// TIA Portal project "Project4" (V18)

(* hardware
DEVICE "S7-1500/ET200MP station_1"  S7-1500 station
   slot 0: "Rail_0"  Rack  6ES7 590-1***0-0AA0
   slot 1: "PLC_1"  CPU 1516F-3 PN/DP  6ES7 516-3FN01-0AB0  V2.9
      slot 3: "CPU display_1"  6ES7591-1BA00-0AA0
      slot 32768: "PROFINET interface_1"  X1
         slot 32769: "Port_1"  X1 P1
         slot 32770: "Port_2"  X1 P2
      slot 33024: "PROFINET interface_2"  X2
         slot 33025: "Port_1"  X2 P1
      slot 33280: "DP interface_1"  X3
      slot 34817: "Virtual CP interface port_1"  Virtual CP interface port  Virtual CP interface port
DEVICE "GSD device_1"  GSD.Device.PN
   slot 0: "Rack"  Rack  V1.0
   slot 0: "UR20-FBC-PN-IRT-V2"  UR20-FBC-PN-IRT-V2 Profinet Device  V01.14.00
      slot 0: "UR20-FBC-PN-IRT-V2 Profinet Device"  UR20-FBC-PN-IRT-V2 Profinet Device
      slot 1: "UR20-FBC-PN-IRT Profinet Device"  UR20-FBC-PN-IRT Profinet Device
         slot 1: "Port 1"  Port 1
         slot 2: "Port 2"  Port 2
   slot 1: "UR20-8DO-P_1"  UR20-8DO-P  1315240000
      slot 0: "UR20-8DO-P"  UR20-8DO-P
   slot 2: "UR20-PF-O-1DI-SIL_1"  UR20-PF-O-1DI-SIL  1335030000
      slot 0: "UR20-PF-O-1DI-SIL"  UR20-PF-O-1DI-SIL
   slot 3: "UR20-16DI-P_1"  UR20-16DI-P  1315200000
      slot 0: "UR20-16DI-P"  UR20-16DI-P
   slot 4: "UR20-4AI-UI-16_1"  UR20-4AI-UI-16  1315620000
      slot 0: "UR20-4AI-UI-16"  UR20-4AI-UI-16
   slot 5: "UR20-4COM-IOL-128BYTE-INOUT_1"  UR20-4COM-IOL-128BYTE-INOUT  1315740000
      slot 0: "UR20-4COM-IOL-128BYTE-INOUT"  UR20-4COM-IOL-128BYTE-INOUT
*)

// ===== PLC "PLC_1"  CPU 1516F-3 PN/DP =====

VAR_GLOBAL   // PLC tag table "Default tag table"
   "UR20_Port0_IN" AT %I16.0 : "DUT_32Bytes";
   "UR20_Port0_OUT" AT %Q16.0 : "DUT_1Bytes";
   "UR20_Port2_OUT" AT %Q17.0 : "DUT_1Bytes";
   "UR20_Port3_OUT" AT %Q18.0 : "DUT_2Bytes";
   "UR20_Port1_IN" AT %I48.0 : "DUT_32Bytes";
   "UR20_Port2_IN" AT %I80.0 : "DUT_32Bytes";
   "UR20_Port3_IN" AT %I112.0 : "DUT_32Bytes";
   "UR20_DIs" AT %I14.0 : "DUT_UR20_DI";
   "UR20_DOs" AT %Q14.0 : "DUT_UR20_DO";
END_VAR

TYPE "DUT_OMRON_E3AS_HL500LMN_IN_Status"
   STRUCT
      ControlOutput1 : Bool;
      ControlOutput2 : Bool;
      InstabilityAlarm : Bool;
      InsufficinetError : Bool;
      Warning : Bool;
      Error : Bool;
   END_STRUCT;
END_TYPE

TYPE "DUT_OMRON_E3AS_HL500LMN_IN"
   STRUCT
      DetectValue : Int;
      LightLevel : Int;
      Status : "DUT_OMRON_E3AS_HL500LMN_IN_Status";
   END_STRUCT;
END_TYPE

TYPE "DUT_NASS_IN"
   STRUCT
      ValveState : Bool;
      ShortCircuit : Bool;
      OpenCircuit : Bool;
      OverHeat : Bool;
      OverCurrent : Bool;
      Counter1OverRun : Bool;
      Counter2OverRun : Bool;
   END_STRUCT;
END_TYPE

TYPE "DUT_NASS_OUT"
   STRUCT
      ON : Bool;
      PWM : Int;
   END_STRUCT;
END_TYPE

TYPE "DUT_OMRON_E2E_X3B4_IL3_2M_IN_Status"
   STRUCT
      Output : Bool;
      Unstable : Bool;
      TooClose : Bool;
      Error : Bool;
   END_STRUCT;
END_TYPE

TYPE "DUT_OMRON_E2E_X3B4_IL3_2M_IN"
   STRUCT
      Montior : Int;
      Status : "DUT_OMRON_E2E_X3B4_IL3_2M_IN_Status";
   END_STRUCT;
END_TYPE

TYPE "DUT_1Bytes"
   STRUCT
      raw : Array[0..0] of Byte;
   END_STRUCT;
END_TYPE

TYPE "DUT_NASS"
   STRUCT
      in : "DUT_NASS_IN";
      out : "DUT_NASS_OUT";
   END_STRUCT;
END_TYPE

TYPE "DUT_2Bytes"
   STRUCT
      raw : Array[0..1] of Byte;
   END_STRUCT;
END_TYPE

TYPE "DUT_4Bytes"
   STRUCT
      raw : Array[0..3] of Byte;
   END_STRUCT;
END_TYPE

TYPE "DUT_32Bytes"
   STRUCT
      raw : Array[0..31] of Byte;
   END_STRUCT;
END_TYPE

TYPE "DUT_UR20_DI"
   STRUCT
      DI1 : Bool;
      DI2 : Bool;
      DI3 : Bool;
      DI4 : Bool;
      CQ1 : Bool;
      CQ2 : Bool;
      CQ3 : Bool;
      CQ4 : Bool;
      ProcessDataInVaildPort1 : Bool;
      ProcessDataInVaildPort2 : Bool;
      ProcessDataInVaildPort3 : Bool;
      ProcessDataInVaildPort4 : Bool;
      ErrorPort1 : Bool;
      ErrorPort2 : Bool;
      ErrorPort3 : Bool;
      ErrorPort4 : Bool;
   END_STRUCT;
END_TYPE

TYPE "DUT_UR20_DO"
   STRUCT
      DO1 : Bool;
      DO2 : Bool;
      DO3 : Bool;
      DO4 : Bool;
      _1 : Bool;
      _2 : Bool;
      _3 : Bool;
      _4 : Bool;
      ProcessDataOutVaildPort1 : Bool;
      ProcessDataOutVaildPort2 : Bool;
      ProcessDataOutVaildPort3 : Bool;
      ProcessDataOutVaildPort4 : Bool;
      _11 : Bool;
      _12 : Bool;
      _13 : Bool;
      _14 : Bool;
   END_STRUCT;
END_TYPE

TYPE "DUT_Murr_59507_OUT"
   STRUCT
      Pin4_X0 : Bool;
      Pin4_X1 : Bool;
      Pin4_X2 : Bool;
      Pin4_X3 : Bool;
      Pin4_X4 : Bool;
      Pin4_X5 : Bool;
      Pin4_X6 : Bool;
      Pin4_X7 : Bool;
   END_STRUCT;
END_TYPE

TYPE "DUT_Murr_59507"
   STRUCT
      in : "DUT_Murr_59507_IN";
      out : "DUT_Murr_59507_OUT";
   END_STRUCT;
END_TYPE

TYPE "DUT_Murr_59507_IN"
   STRUCT
      Pin4_X0 : Bool;
      Pin4_X1 : Bool;
      Pin4_X2 : Bool;
      Pin4_X3 : Bool;
      Pin4_X4 : Bool;
      Pin4_X5 : Bool;
      Pin4_X6 : Bool;
      Pin4_X7 : Bool;
      ErrorPowerSupply : Bool;
      ErrorTemperatureRating : Bool;
      ErrorInputOutput : Bool;
      DIAs : Byte;
      GlobalStatus : Bool;
      DeviceDefine : Byte;
   END_STRUCT;
END_TYPE

DATA_BLOCK "Main_Safety_RTG1_DB"   // DB1, F_DB
{ S7_Optimized_Access := 'TRUE' }
NAME : FUSI
VERSION : 0.1
// stored: InstanceOfName Main_Safety_RTG1
"Main_Safety_RTG1"
BEGIN
END_DATA_BLOCK

DATA_BLOCK "DB_UR20"   // DB2
{ S7_Optimized_Access := 'TRUE' }
VERSION : 0.1
   VAR
      DI : "DUT_UR20_DI";
      "DO" : "DUT_UR20_DO";
      Port0 : "DUT_OMRON_E3AS_HL500LMN_IN";
      Port1 : "DUT_OMRON_E2E_X3B4_IL3_2M_IN";
      Port2 : "DUT_NASS";
      Port3 : "DUT_Murr_59507";
   END_VAR
BEGIN
END_DATA_BLOCK

DATA_BLOCK "FB_UR20_DB"   // DB3
{ S7_Optimized_Access := 'TRUE' }
VERSION : 0.1
// stored: InstanceOfName FB_UR20_IOLINK
"FB_UR20_IOLINK"
BEGIN
END_DATA_BLOCK

DATA_BLOCK "FB_TestFlow_DB"   // DB4
{ S7_Optimized_Access := 'TRUE' }
VERSION : 0.1
// stored: InstanceOfName FB_TestFlow
"FB_TestFlow"
BEGIN
END_DATA_BLOCK

FUNCTION_BLOCK "Main_Safety_RTG1"   // FB1, F_FBD
{ S7_Optimized_Access := 'TRUE' }
BEGIN
END_FUNCTION_BLOCK

FUNCTION_BLOCK "FB_NASS_SmartConnector"   // FB2, LAD
{ S7_Optimized_Access := 'TRUE' }
VERSION : 0.1
   VAR_INPUT
      iEnable : Bool;
   END_VAR
   VAR_IN_OUT
      ioRawIN : Array[*] of Byte;
      ioRawOut : Array[*] of Byte;
      ioData : "DUT_NASS";
   END_VAR
   VAR_TEMP
      _Enable : Bool;
   END_VAR
   VAR_TEMP   // added for the SCL form of the ladder/FBD networks
      _w1 : Bool;
   END_VAR
BEGIN

REGION Network 1
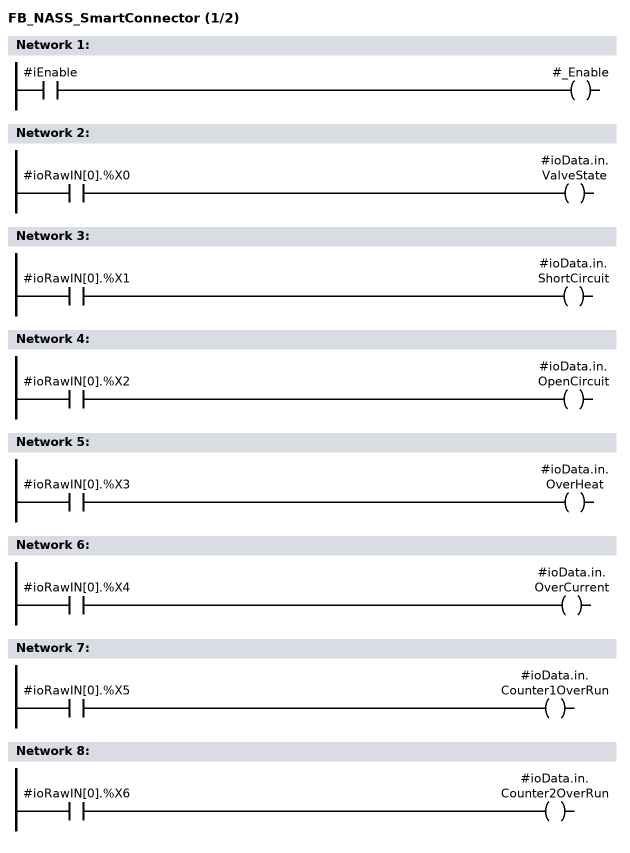
   RUNG wire#powerrail
      Contact( #iEnable )
      Coil( #_Enable )
   END_RUNG
   // the same network as SCL:
   #_Enable := #iEnable;
END_REGION

REGION Network 2
   RUNG wire#powerrail
      Contact( #ioRawIN[0].%X0 )
      Coil( #ioData.in.ValveState )
   END_RUNG
   // the same network as SCL:
   #ioData.in.ValveState := #ioRawIN[0].%X0;
END_REGION

REGION Network 3
   RUNG wire#powerrail
      Contact( #ioRawIN[0].%X1 )
      Coil( #ioData.in.ShortCircuit )
   END_RUNG
   // the same network as SCL:
   #ioData.in.ShortCircuit := #ioRawIN[0].%X1;
END_REGION

REGION Network 4
   RUNG wire#powerrail
      Contact( #ioRawIN[0].%X2 )
      Coil( #ioData.in.OpenCircuit )
   END_RUNG
   // the same network as SCL:
   #ioData.in.OpenCircuit := #ioRawIN[0].%X2;
END_REGION

REGION Network 5
   RUNG wire#powerrail
      Contact( #ioRawIN[0].%X3 )
      Coil( #ioData.in.OverHeat )
   END_RUNG
   // the same network as SCL:
   #ioData.in.OverHeat := #ioRawIN[0].%X3;
END_REGION

REGION Network 6
   RUNG wire#powerrail
      Contact( #ioRawIN[0].%X4 )
      Coil( #ioData.in.OverCurrent )
   END_RUNG
   // the same network as SCL:
   #ioData.in.OverCurrent := #ioRawIN[0].%X4;
END_REGION

REGION Network 7
   RUNG wire#powerrail
      Contact( #ioRawIN[0].%X5 )
      Coil( #ioData.in.Counter1OverRun )
   END_RUNG
   // the same network as SCL:
   #ioData.in.Counter1OverRun := #ioRawIN[0].%X5;
END_REGION

REGION Network 8
   RUNG wire#powerrail
      Contact( #ioRawIN[0].%X6 )
      Coil( #ioData.in.Counter2OverRun )
   END_RUNG
   // the same network as SCL:
   #ioData.in.Counter2OverRun := #ioRawIN[0].%X6;
END_REGION

REGION Network 9
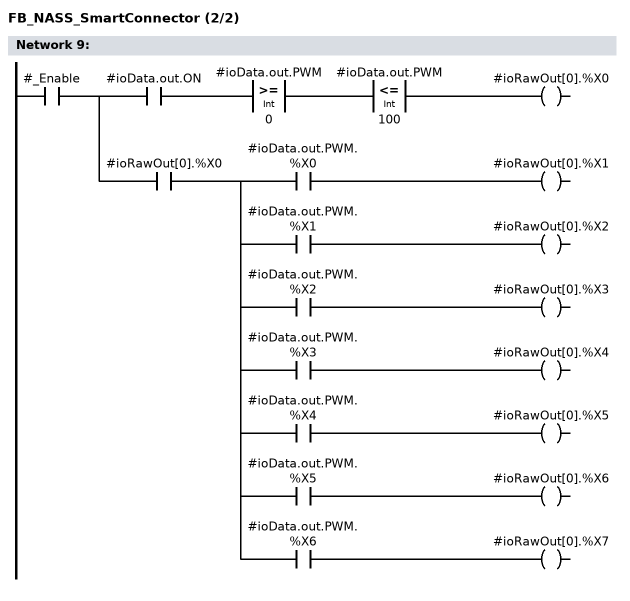
   RUNG wire#powerrail
      Contact( #_Enable )
      wire#w1
      Contact( #ioData.out.ON )
      { S7_Templates := "SrcType := Int" } GE_Contact(in1 := #ioData.out.PWM, in2 := 0)
      { S7_Templates := "SrcType := Int" } LE_Contact(in1 := #ioData.out.PWM, in2 := 100)
      Coil( #ioRawOut[0].%X0 )
   END_RUNG
   RUNG wire#w1
      Contact( #ioRawOut[0].%X0 )
      wire#w2
      Contact( #ioData.out.PWM.%X0 )
      Coil( #ioRawOut[0].%X1 )
   END_RUNG
   RUNG wire#w2
      Contact( #ioData.out.PWM.%X1 )
      Coil( #ioRawOut[0].%X2 )
   END_RUNG
   RUNG wire#w2
      Contact( #ioData.out.PWM.%X2 )
      Coil( #ioRawOut[0].%X3 )
   END_RUNG
   RUNG wire#w2
      Contact( #ioData.out.PWM.%X3 )
      Coil( #ioRawOut[0].%X4 )
   END_RUNG
   RUNG wire#w2
      Contact( #ioData.out.PWM.%X4 )
      Coil( #ioRawOut[0].%X5 )
   END_RUNG
   RUNG wire#w2
      Contact( #ioData.out.PWM.%X5 )
      Coil( #ioRawOut[0].%X6 )
   END_RUNG
   RUNG wire#w2
      Contact( #ioData.out.PWM.%X6 )
      Coil( #ioRawOut[0].%X7 )
   END_RUNG
   // the same network as SCL:
   #ioRawOut[0].%X0 := #_Enable AND #ioData.out.ON AND (#ioData.out.PWM >= 0) AND (#ioData.out.PWM <= 100);
   #_w1 := #_Enable AND #ioRawOut[0].%X0;
   #ioRawOut[0].%X1 := #_w1 AND #ioData.out.PWM.%X0;
   #ioRawOut[0].%X2 := #_w1 AND #ioData.out.PWM.%X1;
   #ioRawOut[0].%X3 := #_w1 AND #ioData.out.PWM.%X2;
   #ioRawOut[0].%X4 := #_w1 AND #ioData.out.PWM.%X3;
   #ioRawOut[0].%X5 := #_w1 AND #ioData.out.PWM.%X4;
   #ioRawOut[0].%X6 := #_w1 AND #ioData.out.PWM.%X5;
   #ioRawOut[0].%X7 := #_w1 AND #ioData.out.PWM.%X6;
END_REGION
END_FUNCTION_BLOCK

FUNCTION_BLOCK "FB_UR20_IOLINK"   // FB3, LAD
{ S7_Optimized_Access := 'TRUE' }
VERSION : 0.1
   VAR
      NassConnector : "FB_NASS_SmartConnector";
      Murr59507 : "FB_Murr_59507";
      OMRONE3ASHL500LMN : "FB_OMRON_E3AS_HL500LMN";
      OMRONE2EX3B4IL32M : "FB_OMRON_E2E_X3B4_IL3_2M";
   END_VAR
   VAR_TEMP
      _temp : Array[0..1] of Byte;
   END_VAR
BEGIN

REGION Network 1
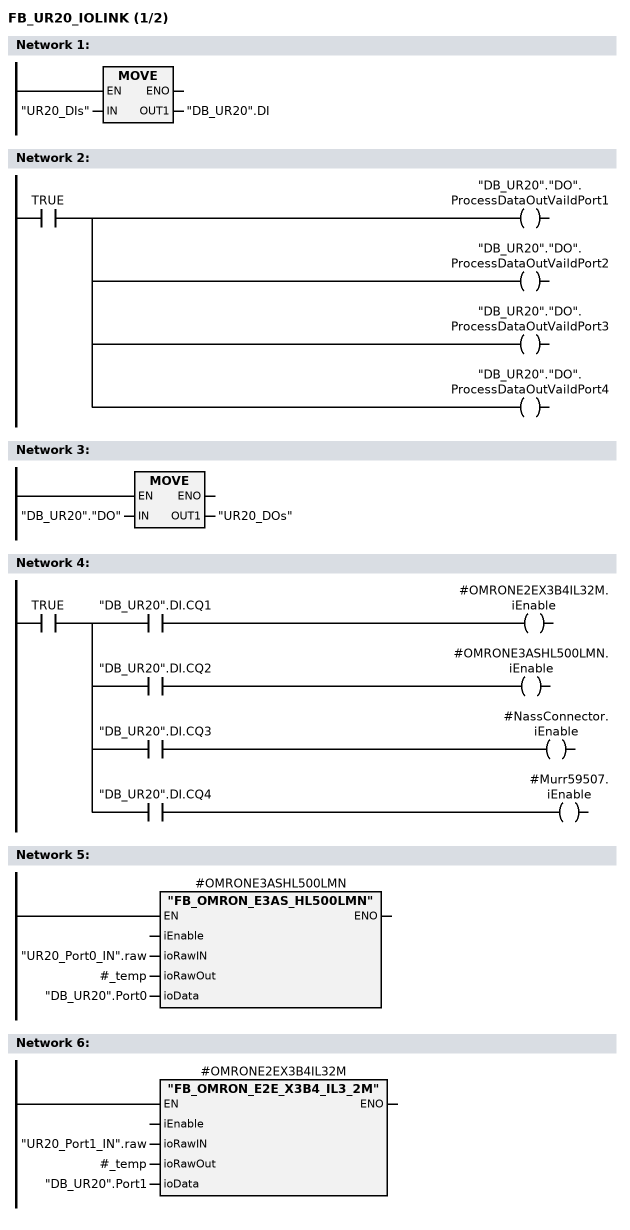
   RUNG wire#powerrail
      Move(in := "UR20_DIs", out1 => "DB_UR20".DI)
   END_RUNG
   // the same network as SCL:
   "DB_UR20".DI := "UR20_DIs";
END_REGION

REGION Network 2
   RUNG wire#powerrail
      Contact( TRUE )
      wire#w1
      Coil( "DB_UR20"."DO".ProcessDataOutVaildPort1 )
   END_RUNG
   RUNG wire#w1
      Coil( "DB_UR20"."DO".ProcessDataOutVaildPort2 )
   END_RUNG
   RUNG wire#w1
      Coil( "DB_UR20"."DO".ProcessDataOutVaildPort3 )
   END_RUNG
   RUNG wire#w1
      Coil( "DB_UR20"."DO".ProcessDataOutVaildPort4 )
   END_RUNG
   // the same network as SCL:
   "DB_UR20"."DO".ProcessDataOutVaildPort1 := TRUE;
   "DB_UR20"."DO".ProcessDataOutVaildPort2 := TRUE;
   "DB_UR20"."DO".ProcessDataOutVaildPort3 := TRUE;
   "DB_UR20"."DO".ProcessDataOutVaildPort4 := TRUE;
END_REGION

REGION Network 3
   RUNG wire#powerrail
      Move(in := "DB_UR20"."DO", out1 => "UR20_DOs")
   END_RUNG
   // the same network as SCL:
   "UR20_DOs" := "DB_UR20"."DO";
END_REGION

REGION Network 4
   RUNG wire#powerrail
      Contact( TRUE )
      wire#w1
      Contact( "DB_UR20".DI.CQ1 )
      Coil( #OMRONE2EX3B4IL32M.iEnable )
   END_RUNG
   RUNG wire#w1
      Contact( "DB_UR20".DI.CQ2 )
      Coil( #OMRONE3ASHL500LMN.iEnable )
   END_RUNG
   RUNG wire#w1
      Contact( "DB_UR20".DI.CQ3 )
      Coil( #NassConnector.iEnable )
   END_RUNG
   RUNG wire#w1
      Contact( "DB_UR20".DI.CQ4 )
      Coil( #Murr59507.iEnable )
   END_RUNG
   // the same network as SCL:
   #OMRONE2EX3B4IL32M.iEnable := TRUE AND "DB_UR20".DI.CQ1;
   #OMRONE3ASHL500LMN.iEnable := TRUE AND "DB_UR20".DI.CQ2;
   #NassConnector.iEnable := TRUE AND "DB_UR20".DI.CQ3;
   #Murr59507.iEnable := TRUE AND "DB_UR20".DI.CQ4;
END_REGION

REGION Network 5
   RUNG wire#powerrail
      #OMRONE3ASHL500LMN(iEnable :=, ioRawIN := "UR20_Port0_IN".raw, ioRawOut := #_temp, ioData := "DB_UR20".Port0)
   END_RUNG
   // the same network as SCL:
   #OMRONE3ASHL500LMN(ioRawIN := "UR20_Port0_IN".raw, ioRawOut := #_temp, ioData := "DB_UR20".Port0);   // "FB_OMRON_E3AS_HL500LMN"
END_REGION

REGION Network 6
   RUNG wire#powerrail
      #OMRONE2EX3B4IL32M(iEnable :=, ioRawIN := "UR20_Port1_IN".raw, ioRawOut := #_temp, ioData := "DB_UR20".Port1)
   END_RUNG
   // the same network as SCL:
   #OMRONE2EX3B4IL32M(ioRawIN := "UR20_Port1_IN".raw, ioRawOut := #_temp, ioData := "DB_UR20".Port1);   // "FB_OMRON_E2E_X3B4_IL3_2M"
END_REGION

REGION Network 7
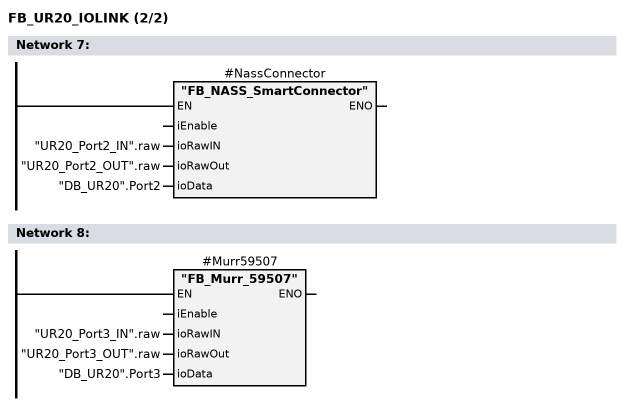
   RUNG wire#powerrail
      #NassConnector(iEnable :=, ioRawIN := "UR20_Port2_IN".raw, ioRawOut := "UR20_Port2_OUT".raw, ioData := "DB_UR20".Port2)
   END_RUNG
   // the same network as SCL:
   #NassConnector(ioRawIN := "UR20_Port2_IN".raw, ioRawOut := "UR20_Port2_OUT".raw, ioData := "DB_UR20".Port2);   // "FB_NASS_SmartConnector"
END_REGION

REGION Network 8
   RUNG wire#powerrail
      #Murr59507(iEnable :=, ioRawIN := "UR20_Port3_IN".raw, ioRawOut := "UR20_Port3_OUT".raw, ioData := "DB_UR20".Port3)
   END_RUNG
   // the same network as SCL:
   #Murr59507(ioRawIN := "UR20_Port3_IN".raw, ioRawOut := "UR20_Port3_OUT".raw, ioData := "DB_UR20".Port3);   // "FB_Murr_59507"
END_REGION
END_FUNCTION_BLOCK

FUNCTION_BLOCK "FB_Murr_59507"   // FB4, LAD
{ S7_Optimized_Access := 'TRUE' }
VERSION : 0.1
   VAR_INPUT
      iEnable : Bool := false;
   END_VAR
   VAR_IN_OUT
      ioRawIN : Array[*] of Byte;
      ioRawOut : Array[*] of Byte;
      ioData : "DUT_Murr_59507";
   END_VAR
   VAR_TEMP
      _Enable : Bool;
   END_VAR
   VAR CONSTANT
      AlwaysON : Bool := 1;
   END_VAR
BEGIN

REGION Network 1
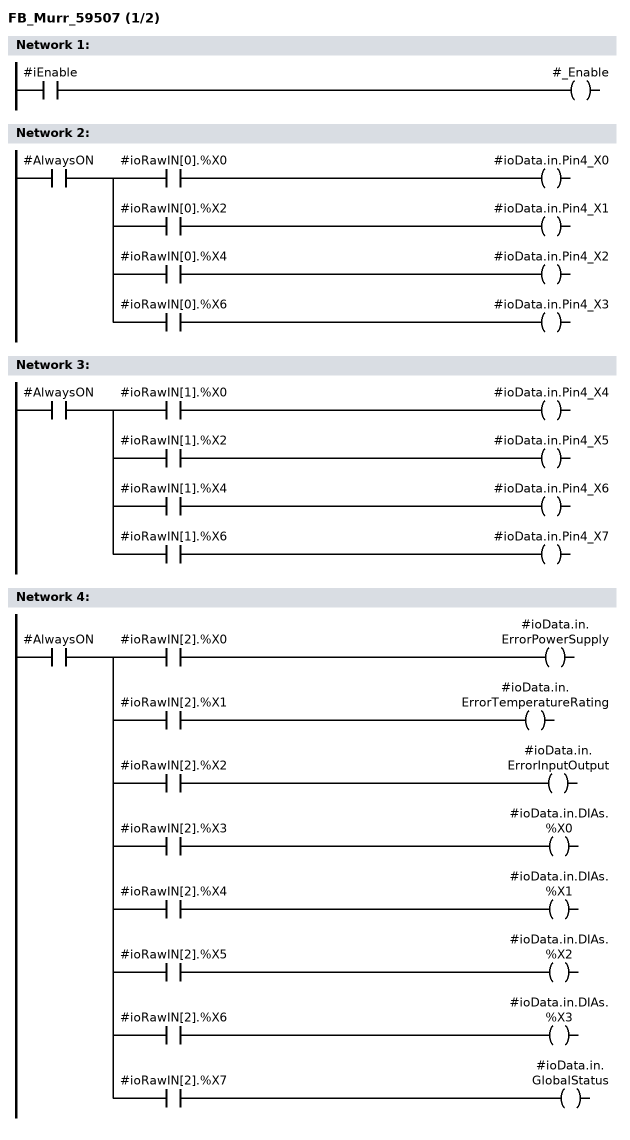
   RUNG wire#powerrail
      Contact( #iEnable )
      Coil( #_Enable )
   END_RUNG
   // the same network as SCL:
   #_Enable := #iEnable;
END_REGION

REGION Network 2
   RUNG wire#powerrail
      Contact( #AlwaysON )
      wire#w1
      Contact( #ioRawIN[0].%X0 )
      Coil( #ioData.in.Pin4_X0 )
   END_RUNG
   RUNG wire#w1
      Contact( #ioRawIN[0].%X2 )
      Coil( #ioData.in.Pin4_X1 )
   END_RUNG
   RUNG wire#w1
      Contact( #ioRawIN[0].%X4 )
      Coil( #ioData.in.Pin4_X2 )
   END_RUNG
   RUNG wire#w1
      Contact( #ioRawIN[0].%X6 )
      Coil( #ioData.in.Pin4_X3 )
   END_RUNG
   // the same network as SCL:
   #ioData.in.Pin4_X0 := #AlwaysON AND #ioRawIN[0].%X0;
   #ioData.in.Pin4_X1 := #AlwaysON AND #ioRawIN[0].%X2;
   #ioData.in.Pin4_X2 := #AlwaysON AND #ioRawIN[0].%X4;
   #ioData.in.Pin4_X3 := #AlwaysON AND #ioRawIN[0].%X6;
END_REGION

REGION Network 3
   RUNG wire#powerrail
      Contact( #AlwaysON )
      wire#w1
      Contact( #ioRawIN[1].%X0 )
      Coil( #ioData.in.Pin4_X4 )
   END_RUNG
   RUNG wire#w1
      Contact( #ioRawIN[1].%X2 )
      Coil( #ioData.in.Pin4_X5 )
   END_RUNG
   RUNG wire#w1
      Contact( #ioRawIN[1].%X4 )
      Coil( #ioData.in.Pin4_X6 )
   END_RUNG
   RUNG wire#w1
      Contact( #ioRawIN[1].%X6 )
      Coil( #ioData.in.Pin4_X7 )
   END_RUNG
   // the same network as SCL:
   #ioData.in.Pin4_X4 := #AlwaysON AND #ioRawIN[1].%X0;
   #ioData.in.Pin4_X5 := #AlwaysON AND #ioRawIN[1].%X2;
   #ioData.in.Pin4_X6 := #AlwaysON AND #ioRawIN[1].%X4;
   #ioData.in.Pin4_X7 := #AlwaysON AND #ioRawIN[1].%X6;
END_REGION

REGION Network 4
   RUNG wire#powerrail
      Contact( #AlwaysON )
      wire#w1
      Contact( #ioRawIN[2].%X0 )
      Coil( #ioData.in.ErrorPowerSupply )
   END_RUNG
   RUNG wire#w1
      Contact( #ioRawIN[2].%X1 )
      Coil( #ioData.in.ErrorTemperatureRating )
   END_RUNG
   RUNG wire#w1
      Contact( #ioRawIN[2].%X2 )
      Coil( #ioData.in.ErrorInputOutput )
   END_RUNG
   RUNG wire#w1
      Contact( #ioRawIN[2].%X3 )
      Coil( #ioData.in.DIAs.%X0 )
   END_RUNG
   RUNG wire#w1
      Contact( #ioRawIN[2].%X4 )
      Coil( #ioData.in.DIAs.%X1 )
   END_RUNG
   RUNG wire#w1
      Contact( #ioRawIN[2].%X5 )
      Coil( #ioData.in.DIAs.%X2 )
   END_RUNG
   RUNG wire#w1
      Contact( #ioRawIN[2].%X6 )
      Coil( #ioData.in.DIAs.%X3 )
   END_RUNG
   RUNG wire#w1
      Contact( #ioRawIN[2].%X7 )
      Coil( #ioData.in.GlobalStatus )
   END_RUNG
   // the same network as SCL:
   #ioData.in.ErrorPowerSupply := #AlwaysON AND #ioRawIN[2].%X0;
   #ioData.in.ErrorTemperatureRating := #AlwaysON AND #ioRawIN[2].%X1;
   #ioData.in.ErrorInputOutput := #AlwaysON AND #ioRawIN[2].%X2;
   #ioData.in.DIAs.%X0 := #AlwaysON AND #ioRawIN[2].%X3;
   #ioData.in.DIAs.%X1 := #AlwaysON AND #ioRawIN[2].%X4;
   #ioData.in.DIAs.%X2 := #AlwaysON AND #ioRawIN[2].%X5;
   #ioData.in.DIAs.%X3 := #AlwaysON AND #ioRawIN[2].%X6;
   #ioData.in.GlobalStatus := #AlwaysON AND #ioRawIN[2].%X7;
END_REGION

REGION Network 5
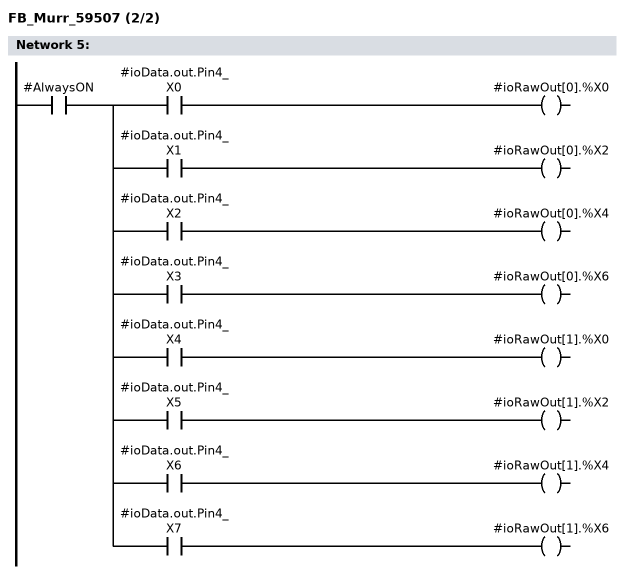
   RUNG wire#powerrail
      Contact( #AlwaysON )
      wire#w1
      Contact( #ioData.out.Pin4_X0 )
      Coil( #ioRawOut[0].%X0 )
   END_RUNG
   RUNG wire#w1
      Contact( #ioData.out.Pin4_X1 )
      Coil( #ioRawOut[0].%X2 )
   END_RUNG
   RUNG wire#w1
      Contact( #ioData.out.Pin4_X2 )
      Coil( #ioRawOut[0].%X4 )
   END_RUNG
   RUNG wire#w1
      Contact( #ioData.out.Pin4_X3 )
      Coil( #ioRawOut[0].%X6 )
   END_RUNG
   RUNG wire#w1
      Contact( #ioData.out.Pin4_X4 )
      Coil( #ioRawOut[1].%X0 )
   END_RUNG
   RUNG wire#w1
      Contact( #ioData.out.Pin4_X5 )
      Coil( #ioRawOut[1].%X2 )
   END_RUNG
   RUNG wire#w1
      Contact( #ioData.out.Pin4_X6 )
      Coil( #ioRawOut[1].%X4 )
   END_RUNG
   RUNG wire#w1
      Contact( #ioData.out.Pin4_X7 )
      Coil( #ioRawOut[1].%X6 )
   END_RUNG
   // the same network as SCL:
   #ioRawOut[0].%X0 := #AlwaysON AND #ioData.out.Pin4_X0;
   #ioRawOut[0].%X2 := #AlwaysON AND #ioData.out.Pin4_X1;
   #ioRawOut[0].%X4 := #AlwaysON AND #ioData.out.Pin4_X2;
   #ioRawOut[0].%X6 := #AlwaysON AND #ioData.out.Pin4_X3;
   #ioRawOut[1].%X0 := #AlwaysON AND #ioData.out.Pin4_X4;
   #ioRawOut[1].%X2 := #AlwaysON AND #ioData.out.Pin4_X5;
   #ioRawOut[1].%X4 := #AlwaysON AND #ioData.out.Pin4_X6;
   #ioRawOut[1].%X6 := #AlwaysON AND #ioData.out.Pin4_X7;
END_REGION
END_FUNCTION_BLOCK

FUNCTION_BLOCK "FB_OMRON_E3AS_HL500LMN"   // FB5, LAD
{ S7_Optimized_Access := 'TRUE' }
VERSION : 0.1
   VAR_INPUT
      iEnable : Bool;
   END_VAR
   VAR_IN_OUT
      ioRawIN : Array[*] of Byte;
      ioRawOut : Array[*] of Byte;
      ioData : "DUT_OMRON_E3AS_HL500LMN_IN";
   END_VAR
   VAR_TEMP
      _Enable : Bool;
   END_VAR
   VAR CONSTANT
      AlwaysON : Bool := 1;
   END_VAR
BEGIN

REGION Network 1
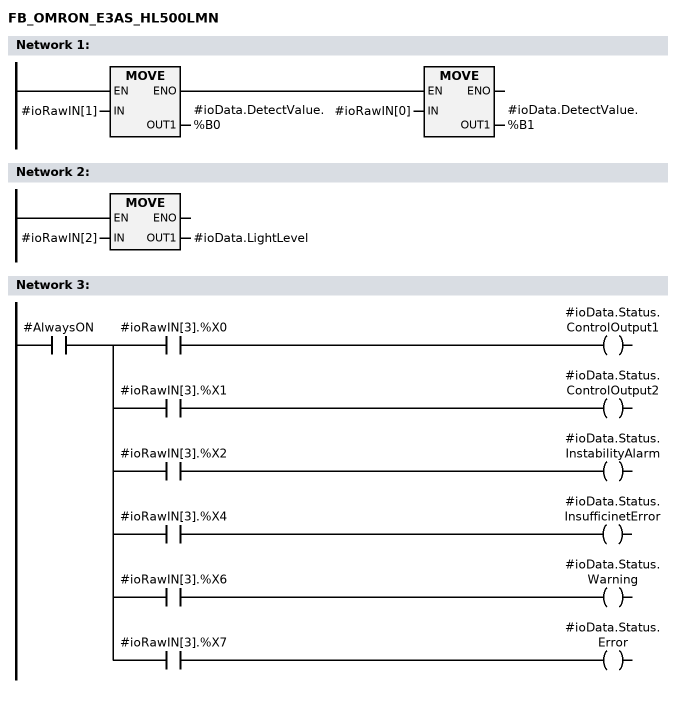
   RUNG wire#powerrail
      Move(in := #ioRawIN[1], out1 => #ioData.DetectValue.%B0)
      Move(in := #ioRawIN[0], out1 => #ioData.DetectValue.%B1)
   END_RUNG
   // the same network as SCL:
   #ioData.DetectValue.%B0 := #ioRawIN[1];
   #ioData.DetectValue.%B1 := #ioRawIN[0];
END_REGION

REGION Network 2
   RUNG wire#powerrail
      Move(in := #ioRawIN[2], out1 => #ioData.LightLevel)
   END_RUNG
   // the same network as SCL:
   #ioData.LightLevel := #ioRawIN[2];
END_REGION

REGION Network 3
   RUNG wire#powerrail
      Contact( #AlwaysON )
      wire#w1
      Contact( #ioRawIN[3].%X0 )
      Coil( #ioData.Status.ControlOutput1 )
   END_RUNG
   RUNG wire#w1
      Contact( #ioRawIN[3].%X1 )
      Coil( #ioData.Status.ControlOutput2 )
   END_RUNG
   RUNG wire#w1
      Contact( #ioRawIN[3].%X2 )
      Coil( #ioData.Status.InstabilityAlarm )
   END_RUNG
   RUNG wire#w1
      Contact( #ioRawIN[3].%X4 )
      Coil( #ioData.Status.InsufficinetError )
   END_RUNG
   RUNG wire#w1
      Contact( #ioRawIN[3].%X6 )
      Coil( #ioData.Status.Warning )
   END_RUNG
   RUNG wire#w1
      Contact( #ioRawIN[3].%X7 )
      Coil( #ioData.Status.Error )
   END_RUNG
   // the same network as SCL:
   #ioData.Status.ControlOutput1 := #AlwaysON AND #ioRawIN[3].%X0;
   #ioData.Status.ControlOutput2 := #AlwaysON AND #ioRawIN[3].%X1;
   #ioData.Status.InstabilityAlarm := #AlwaysON AND #ioRawIN[3].%X2;
   #ioData.Status.InsufficinetError := #AlwaysON AND #ioRawIN[3].%X4;
   #ioData.Status.Warning := #AlwaysON AND #ioRawIN[3].%X6;
   #ioData.Status.Error := #AlwaysON AND #ioRawIN[3].%X7;
END_REGION
END_FUNCTION_BLOCK

FUNCTION_BLOCK "FB_OMRON_E2E_X3B4_IL3_2M"   // FB6, LAD
{ S7_Optimized_Access := 'TRUE' }
VERSION : 0.1
   VAR_INPUT
      iEnable : Bool := false;
   END_VAR
   VAR_IN_OUT
      ioRawIN : Array[*] of Byte;
      ioRawOut : Array[*] of Byte;
      ioData : "DUT_OMRON_E2E_X3B4_IL3_2M_IN";
   END_VAR
   VAR_TEMP
      _Enable : Bool;
   END_VAR
   VAR CONSTANT
      AlwaysON : Bool := 1;
   END_VAR
BEGIN

REGION Network 1
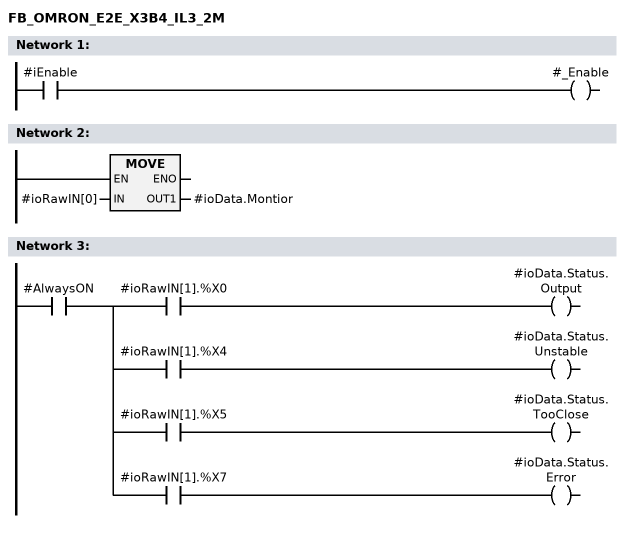
   RUNG wire#powerrail
      Contact( #iEnable )
      Coil( #_Enable )
   END_RUNG
   // the same network as SCL:
   #_Enable := #iEnable;
END_REGION

REGION Network 2
   RUNG wire#powerrail
      Move(in := #ioRawIN[0], out1 => #ioData.Montior)
   END_RUNG
   // the same network as SCL:
   #ioData.Montior := #ioRawIN[0];
END_REGION

REGION Network 3
   RUNG wire#powerrail
      Contact( #AlwaysON )
      wire#w1
      Contact( #ioRawIN[1].%X0 )
      Coil( #ioData.Status.Output )
   END_RUNG
   RUNG wire#w1
      Contact( #ioRawIN[1].%X4 )
      Coil( #ioData.Status.Unstable )
   END_RUNG
   RUNG wire#w1
      Contact( #ioRawIN[1].%X5 )
      Coil( #ioData.Status.TooClose )
   END_RUNG
   RUNG wire#w1
      Contact( #ioRawIN[1].%X7 )
      Coil( #ioData.Status.Error )
   END_RUNG
   // the same network as SCL:
   #ioData.Status.Output := #AlwaysON AND #ioRawIN[1].%X0;
   #ioData.Status.Unstable := #AlwaysON AND #ioRawIN[1].%X4;
   #ioData.Status.TooClose := #AlwaysON AND #ioRawIN[1].%X5;
   #ioData.Status.Error := #AlwaysON AND #ioRawIN[1].%X7;
END_REGION
END_FUNCTION_BLOCK

FUNCTION_BLOCK "FB_TestFlow"   // FB7, GRAPH_PLUS
{ S7_Optimized_Access := 'TRUE' }
VERSION : 0.1
   VAR_INPUT
      OFF_SQ : Bool := false;   // Turn sequence off
      INIT_SQ : Bool := false;   // Set sequence to initial state
      ACK_EF : Bool := false;   // Acknowledge all errors and faults
      S_PREV : Bool := false;   // Output previous step in parameter S_NO
      S_NEXT : Bool := false;   // Indicate next step in parameter S_NO
      SW_AUTO : Bool := false;   // Automatic mode
      SW_TAP : Bool := false;   // Semiautomatic/switch with transition
      SW_TOP : Bool := false;   // Semiautomatic/ignore transition
      SW_MAN : Bool := false;   // Manual mode
      S_SEL : Int := 0;   // Select step to be output to S_NO
      S_ON : Bool := false;   // Activate step indicated in S_NO
      S_OFF : Bool := false;   // Disable step indicated in S_NO
      T_PUSH : Bool := false;   // Enable transition to switch in semi automatic mode
   END_VAR
   VAR_OUTPUT
      S_NO : Int := 0;   // Step number
      S_MORE : Bool := false;   // More steps are available and can be shown in S_NO
      S_ACTIVE : Bool := false;   // Step indicated in S_NO is active
      ERR_FLT : Bool := false;   // Interlock or supervision group error
      AUTO_ON : Bool := false;   // Automatic mode is active
      TAP_ON : Bool := false;   // Semiautomatic mode/step with transition enabled
      TOP_ON : Bool := false;   // Semiautomatic mode/ignore transition enabled
      MAN_ON : Bool := false;   // Manual mode is active
   END_VAR
   VAR
      HMI_INFO : Array[0..10] of UInt;
      IF_PAR : G7_IfParPlus_V6;
      RT_DATA : G7_RTDataPlus_V6;   // Internal data area
      Trans1 : G7_TransitionPlus_V6;   // Transition structure
      Trans3 : G7_TransitionPlus_V6;   // Transition structure
      Trans4 : G7_TransitionPlus_V6;   // Transition structure
      Trans5 : G7_TransitionPlus_V6;   // Transition structure
      Trans6 : G7_TransitionPlus_V6;   // Transition structure
      Trans7 : G7_TransitionPlus_V6;   // Transition structure
      Trans9 : G7_TransitionPlus_V6;   // Transition structure
      Trans10 : G7_TransitionPlus_V6;   // Transition structure
      Trans11 : G7_TransitionPlus_V6;   // Transition structure
      Step1 : G7_StepPlus_V6;   // Step structure
      Step3 : G7_StepPlus_V6;   // Step structure
      Step4 : G7_StepPlus_V6;   // Step structure
      Step5 : G7_StepPlus_V6;   // Step structure
      Step6 : G7_StepPlus_V6;   // Step structure
      Step7 : G7_StepPlus_V6;   // Step structure
      Step8 : G7_StepPlus_V6;   // Step structure
      Step9 : G7_StepPlus_V6;   // Step structure
      Step10 : G7_StepPlus_V6;   // Step structure
      Step11 : G7_StepPlus_V6;   // Step structure
      SINI : Array[0..3] of USInt;
      LSTT : Array[0..8] of USInt;
      ATAJ : Array[0..8] of USInt;
      ATAB : Array[0..8] of USInt;
      PSTT : Array[0..8] of USInt;
      NSTT : Array[0..8] of USInt;
      ASSJ : Array[0..9] of USInt;
      ASSB : Array[0..9] of USInt;
      PTTS : Array[0..9] of USInt;
      NTTS : Array[0..9] of USInt;
      SW_SQTS : Array[0..9] of USInt;
      SWITCH : Array[0..1] of USInt;
      TVX : Array[0..3] of USInt;
      TTX : Array[0..3] of USInt;
      TSX : Array[0..3] of USInt;
      S00X : Array[0..3] of USInt;
      SOFFX : Array[0..3] of USInt;
      SONX : Array[0..3] of USInt;
      SAX : Array[0..3] of USInt;
      SERRX : Array[0..10] of USInt;
      SMX : Array[0..10] of USInt;
      S0X : Array[0..10] of USInt;
      S1X : Array[0..10] of USInt;
      IL_ALARM_INST : Diag_Alarm;
      SUP_ALARM_INST : Diag_Alarm;
      STEP_TIME_ALARM_INST : Diag_Alarm;
      IEC_TIMER_INST : IEC_TIMER;
      TRANSACTION_FLAG : Bool := false;
   END_VAR
   // SINI[0] := 2;
   // LSTT[0] := 255;
   // ATAJ[1] := 1;
   // ATAB[1] := 1;
   // PSTT[1] := 1;
   // NSTT[0] := 1;
   // ASSJ[1] := 1;
   // ASSB[1] := 1;
   // PTTS[0] := 255;
   // NTTS[1] := 1;
   // TVX[0] := 16#1;
   // TTX[0] := 16#1;
   // TSX[0] := 16#1;
   // S00X[0] := 16#1;
   // SOFFX[0] := 16#1;
   // SONX[0] := 16#1;
   // SAX[0] := 16#1;
   // SERRX[0] := 16#1;
   // SMX[0] := 16#1;
   // S0X[0] := 16#1;
   // S1X[0] := 16#1;
   // SINI[2] := 255;
   // SINI[3] := 255;
   // LSTT[1] := 255;
   // LSTT[2] := 255;
   // LSTT[3] := 255;
   // LSTT[4] := 255;
   // LSTT[5] := 255;
   // LSTT[6] := 255;
   // LSTT[8] := 255;
   // ATAJ[2] := 2;
   // ATAJ[3] := 3;
   // ATAJ[4] := 4;
   // ATAJ[5] := 5;
   // ATAJ[6] := 6;
   // ATAJ[7] := 7;
   // ATAJ[8] := 8;
   // ATAB[2] := 2;
   // ATAB[3] := 3;
   // ATAB[4] := 4;
   // ATAB[5] := 5;
   // ATAB[6] := 6;
   // ATAB[7] := 7;
   // ATAB[8] := 8;
   // PSTT[2] := 2;
   // PSTT[3] := 3;
   // PSTT[4] := 4;
   // PSTT[5] := 5;
   // PSTT[6] := 7;
   // PSTT[7] := 8;
   // PSTT[8] := 9;
   // NSTT[1] := 2;
   // NSTT[2] := 3;
   // NSTT[3] := 4;
   // NSTT[4] := 5;
   // NSTT[5] := 7;
   // NSTT[6] := 9;
   // NSTT[8] := 8;
   // ASSJ[2] := 2;
   // ASSJ[3] := 3;
   // ASSJ[4] := 4;
   // ASSJ[5] := 6;
   // ASSJ[6] := 5;
   // ASSJ[7] := 7;
   // ASSJ[8] := 8;
   // ASSJ[9] := 9;
   // ASSB[2] := 2;
   // ASSB[3] := 3;
   // ASSB[4] := 4;
   // ASSB[5] := 6;
   // ASSB[6] := 5;
   // ASSB[7] := 7;
   // ASSB[8] := 8;
   // ASSB[9] := 9;
   // PTTS[2] := 1;
   // PTTS[3] := 2;
   // PTTS[4] := 3;
   // PTTS[5] := 4;
   // PTTS[6] := 4;
   // PTTS[7] := 5;
   // PTTS[8] := 8;
   // PTTS[9] := 6;
   // NTTS[2] := 2;
   // NTTS[3] := 3;
   // NTTS[4] := 4;
   // NTTS[5] := 5;
   // NTTS[6] := 5;
   // NTTS[7] := 6;
   // NTTS[8] := 7;
   // NTTS[9] := 8;
   // SW_SQTS[5] := 1;
   // SW_SQTS[6] := 2;
   // SW_SQTS[7] := 3;
   // SW_SQTS[8] := 3;
   // SW_SQTS[9] := 3;
   // SWITCH[0] := 64;
   // SWITCH[1] := 2;
BEGIN
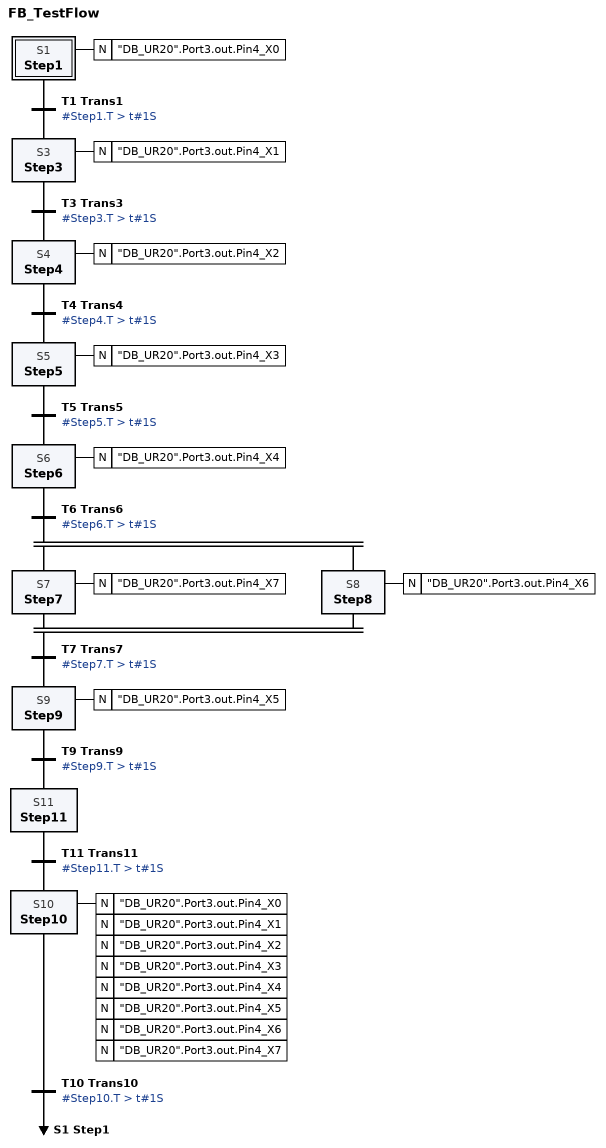
   // sequencer 1
   INITIAL_STEP Step1:   // S1, max time T#10S, warning time T#7S
              N    "DB_UR20".Port3.out.Pin4_X0
   END_STEP
   TRANSITION Trans1 FROM Step1 TO Step3   // T1
      := #Step1.T > t#1S;
   END_TRANSITION
   STEP Step3:   // S3, max time T#10S, warning time T#7S
              N    "DB_UR20".Port3.out.Pin4_X1
   END_STEP
   TRANSITION Trans3 FROM Step3 TO Step4   // T3
      := #Step3.T > t#1S;
   END_TRANSITION
   STEP Step4:   // S4, max time T#10S, warning time T#7S
              N    "DB_UR20".Port3.out.Pin4_X2
   END_STEP
   TRANSITION Trans4 FROM Step4 TO Step5   // T4
      := #Step4.T > t#1S;
   END_TRANSITION
   STEP Step5:   // S5, max time T#10S, warning time T#7S
              N    "DB_UR20".Port3.out.Pin4_X3
   END_STEP
   TRANSITION Trans5 FROM Step5 TO Step6   // T5
      := #Step5.T > t#1S;
   END_TRANSITION
   STEP Step6:   // S6, max time T#10S, warning time T#7S
              N    "DB_UR20".Port3.out.Pin4_X4
   END_STEP
   TRANSITION Trans6 FROM Step6 TO (Step7, Step8)   // T6
      := #Step6.T > t#1S;
   END_TRANSITION
   STEP Step7:   // S7, max time T#10S, warning time T#7S
              N    "DB_UR20".Port3.out.Pin4_X7
   END_STEP
   STEP Step8:   // S8, max time T#10S, warning time T#7S
              N    "DB_UR20".Port3.out.Pin4_X6
   END_STEP
   TRANSITION Trans7 FROM (Step7, Step8) TO Step9   // T7
      := #Step7.T > t#1S;
   END_TRANSITION
   STEP Step9:   // S9, max time T#10S, warning time T#7S
              N    "DB_UR20".Port3.out.Pin4_X5
   END_STEP
   TRANSITION Trans9 FROM Step9 TO Step11   // T9
      := #Step9.T > t#1S;
   END_TRANSITION
   STEP Step10:   // S10, max time T#10S, warning time T#7S
              N    "DB_UR20".Port3.out.Pin4_X0
              N    "DB_UR20".Port3.out.Pin4_X1
              N    "DB_UR20".Port3.out.Pin4_X2
              N    "DB_UR20".Port3.out.Pin4_X3
              N    "DB_UR20".Port3.out.Pin4_X4
              N    "DB_UR20".Port3.out.Pin4_X5
              N    "DB_UR20".Port3.out.Pin4_X6
              N    "DB_UR20".Port3.out.Pin4_X7
   END_STEP
   TRANSITION Trans10 FROM Step10 TO Step1   // T10, jump
      := #Step10.T > t#1S;
   END_TRANSITION
   STEP Step11:   // S11, max time T#10S, warning time T#7S
   END_STEP
   TRANSITION Trans11 FROM Step11 TO Step10   // T11
      := #Step11.T > t#1S;
   END_TRANSITION
END_FUNCTION_BLOCK

ORGANIZATION_BLOCK "Main"   // OB1, LAD, ProgramCycle
TITLE = "Main Program Sweep (Cycle)"
{ S7_Optimized_Access := 'TRUE' }
VERSION : 0.1
   VAR_INPUT
      Initial_Call : Bool;   // Initial call of this OB
      Remanence : Bool;   // =True, if remanent data are available
   END_VAR
BEGIN

REGION Network 1
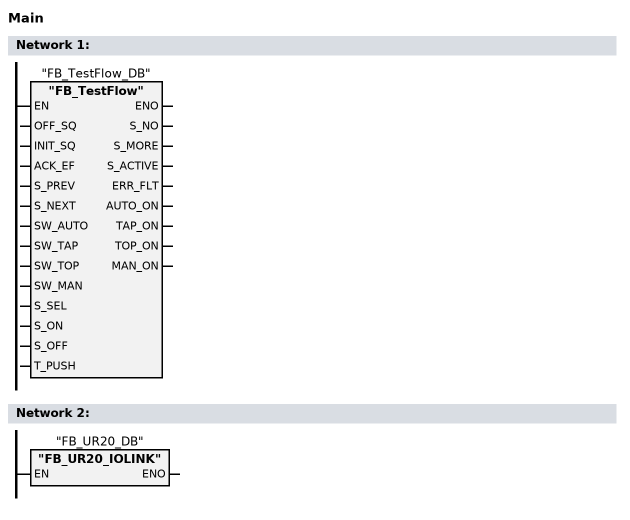
   RUNG wire#powerrail
      "FB_TestFlow_DB"(OFF_SQ :=, INIT_SQ :=, ACK_EF :=, S_PREV :=, S_NEXT :=, SW_AUTO :=, SW_TAP :=, SW_TOP :=, SW_MAN :=, S_SEL :=, S_ON :=, S_OFF :=, T_PUSH :=, S_NO =>, S_MORE =>, S_ACTIVE =>, ERR_FLT =>, AUTO_ON =>, TAP_ON =>, TOP_ON =>, MAN_ON =>)
   END_RUNG
   // the same network as SCL:
   "FB_TestFlow_DB"();   // "FB_TestFlow"
END_REGION

REGION Network 2
   RUNG wire#powerrail
      "FB_UR20_DB"()
   END_RUNG
   // the same network as SCL:
   "FB_UR20_DB"();   // "FB_UR20_IOLINK"
END_REGION
END_ORGANIZATION_BLOCK